PROGRAM MAIN
VAR
END_VAR

END_PROGRAM

(* stored: Version 1.1.0.1
   POU MAIN: Id {4c3786fc-21e7-4a49-a02d-e42936347c82} *)
